{attribute 'GeneratedUsingTerminal: EL5101-0011-0016'}
{attribute addProperty BoxType "EL5101-0011-0016"}
{attribute addProperty Id "ENC_StatusAT %I*ENC_Status_4E2088B98ENC_NextSync1TimeAT %I*ENC_NextSync1Time_9AFDC2758ENC_TxPdo_1_Samples_Counter_valueAT %I*ENC_TxPdo_1_Samples_Counter_value_215818C64ENC_ControlAT %Q*ENC_Control_14E3EF4F5WcStateAT %I*WcState_9091E0EB2InfoDataAT %I*InfoData_1088C70510"}
{attribute addProperty CRC "498427049"}
{attribute addProperty Size "37"}
TYPE EL5101_1DB564A9 EXTENDS EtcSlaveTerminalBase_947E5A46 :
STRUCT
	{attribute addProperty Name "ENC_Status"}
	ENC_Status : ENC_Status_4E2088B9;
	{attribute addProperty Name "ENC_NextSync1Time"}
	ENC_NextSync1Time : ENC_NextSync1Time_9AFDC275;
	{attribute addProperty Name "ENC_TxPdo_1_Samples_Counter_value"}
	ENC_TxPdo_1_Samples_Counter_value : ENC_TxPdo_1_Samples_Counter_value_215818C6;
	{attribute addProperty Name "ENC_Control"}
	ENC_Control : ENC_Control_14E3EF4F;
	{attribute addProperty Name "WcState"}
	WcState : WcState_9091E0EB;
	{attribute addProperty Name "InfoData"}
	InfoData : InfoData_1088C705;
END_STRUCT
END_TYPE

(* stored: Version 1.2.0.0, ProductVersion 3.1.4024.9
   DUT EL5101_1DB564A9: Id {72ddec6d-d54d-4aaf-bb37-49699689e4c0} *)
